DATA_BLOCK "ST10_Flow26_JMagnetLoad&Unload_iDB"
{ S7_Optimized_Access := 'TRUE' }
VERSION : 0.1
NON_RETAIN
// ATTRIBUTES
// AUTO_NUMBER = False
// BLOCK_NUMBER = 1096
// END_ATTRIBUTES
"ST10_Flow26_JMagnetLoad&Unload"

BEGIN

END_DATA_BLOCK

